// TIA Portal V20 export
TYPE "LKinCtrl_typeSettings"
   STRUCT
      kinematics { ExternalAccessible := 'False'; ExternalVisible := 'False'; ExternalWritable := 'False'; S7_SetPoint := 'True'} : "LKinCtrl_typeConfigurationKinematics";
      kinematicAxes { ExternalAccessible := 'False'; ExternalVisible := 'False'; ExternalWritable := 'False'; S7_SetPoint := 'True'} : Array[1.."LKINCTRL_KINEMATICS_AXES"] of "LKinCtrl_typeConfigurationAxis";
      movePathConfiguration { ExternalAccessible := 'False'; ExternalVisible := 'False'; ExternalWritable := 'False'; S7_SetPoint := 'True'} : "LKinCtrl_typeConfiguration";
   END_STRUCT;
END_TYPE
